{attribute 'linkalways'} 
{attribute 'no_explicit_call' := 'This FB is a CLASS and must be accessed using methods or properties'}
{attribute 'enable_dynamic_creation'}
FUNCTION_BLOCK FINAL MAX_LINT EXTENDS Node
VAR
	in1 : _LINT(0);
	in2 : _LINT(0);
	out : _LINT(0);
END_VAR

METHOD PUBLIC Clone : I_Node
VAR
	pNode : POINTER TO MAX_LINT;
END_VAR
pNode := __NEW(MAX_LINT);
Clone := pNode^;
END_METHOD

METHOD FB_init : BOOL
VAR_INPUT
	bInitRetains : BOOL; // if TRUE, the retain variables are initialized (warm start / cold start)
	bInCopyCode : BOOL;  // if TRUE, the instance afterwards gets moved into the copy code (online change)
END_VAR
AddInput('in1',THIS^.in1);
AddInput('in2',THIS^.in2);
AddOutput('out', THIS^.out);
END_METHOD

METHOD PROTECTED OnExecute
VAR
END_VAR
out.Value := MAX(in1.Value, in2.Value);
END_METHOD

END_FUNCTION_BLOCK

(* stored: Version 1.1.0.1, ProductVersion 3.1.4024.15
   POU MAX_LINT: Id {59e9c2ba-2c79-4369-b9b9-ca5f931f5e8d}, SpecialFunc None
   Folder Constructor: Id {d4a2d313-d888-4725-89c9-aad654731a28}
   Method Clone: Id {bf345d08-2893-4c63-96e2-03c997542b11}
   Method FB_init: Id {0e46d78c-2864-432f-abf4-dd2a87d22412}
   Method OnExecute: Id {3d6e61e5-edcc-4b3f-b1ee-9e70a2c677d9} *)
